// Mitsubishi GX Works2 project: Control Status2   PLC: FX1S

PROGRAM MAIN
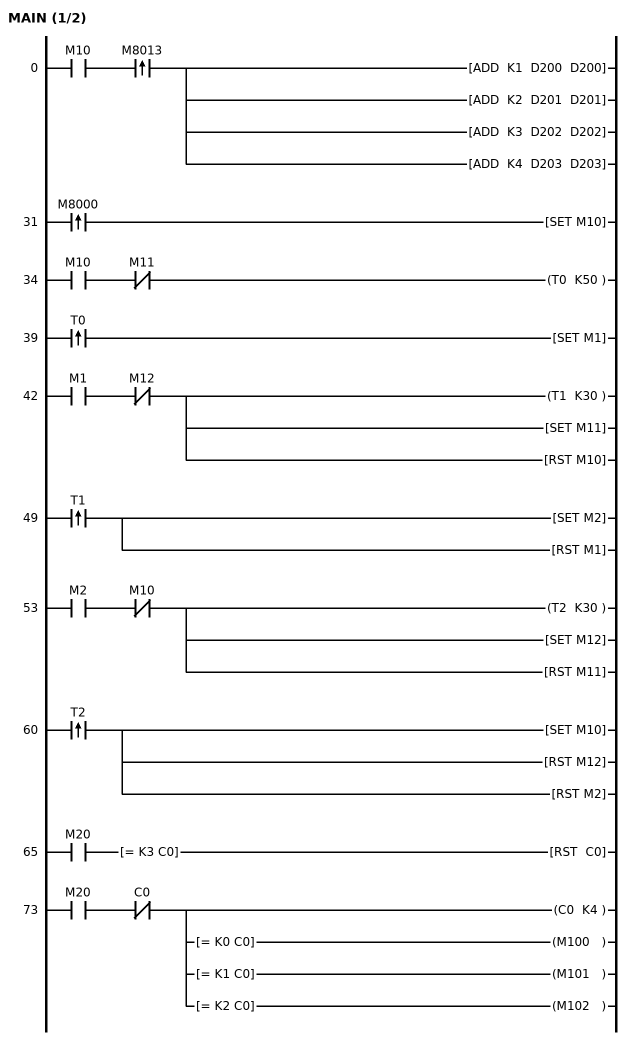
0     LD      M10
      ANDP    M8013
      ADD     K1 D200 D200
      ADD     K2 D201 D201
      ADD     K3 D202 D202
      ADD     K4 D203 D203
31    LDP     M8000
      SET     M10
34    LD      M10
      ANI     M11
      OUT     T0 K50
39    LDP     T0
      SET     M1
42    LD      M1
      ANI     M12
      OUT     T1 K30
      SET     M11
      RST     M10
49    LDP     T1
      SET     M2
      RST     M1
53    LD      M2
      ANI     M10
      OUT     T2 K30
      SET     M12
      RST     M11
60    LDP     T2
      SET     M10
      RST     M12
      RST     M2
65    LD      M20
      AND=    K3 C0
      RST     C0
73    LD      M20
      ANI     C0
      OUT     C0 K4
      MPS
      AND=    K0 C0
      OUT     M100
      MRD
      AND=    K1 C0
      OUT     M101
      MPP
      AND=    K2 C0
      OUT     M102
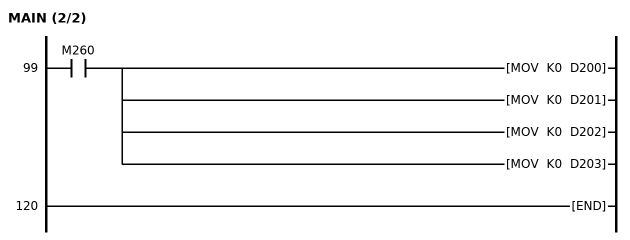
99    LD      M260
      MOV     K0 D200
      MOV     K0 D201
      MOV     K0 D202
      MOV     K0 D203
120   END
END_PROGRAM
